// TIA Portal V15 export
// export: Created 2018-05-29T12:25:38.1552518Z, ExportSetting WithDefaults, DisplayName Totally Integrated Automation Portal, DisplayVersion V15, DisplayName STEP 7 Professional, DisplayVersion V15, DisplayName WinCC Professional, DisplayVersion V15, DisplayName TIA Portal Openness, DisplayVersion V15
FUNCTION "LIC006_fc" : Void   // FC1, STL
TITLE = LIC006_fc
{ S7_Optimized_Access := 'TRUE' }
VERSION : 0.1
// test
// stored: AutoNumber true, UDAEnableTagReadback false
BEGIN

NETWORK
TITLE = Change PID Setpoints
// The phase FBs write on the operator setpoints of the PID-controller
// To avoid that the setpoints are always overwritten (and blocking operator control)
// we use pulses generated by the phase to set the setpoints only at specific moments
// i_fOCmdSP (setpoint)
// i_fOCmdMANOP (output)
      CALL  "BST_PIDAIN_400", "DB";


//Write the Operator_Setpoint
      A     "LIC006_sp".Set_SP;
      JCN   J001;

      L     "LIC006_sp".Operator_Setpoint;
      T     "LIC006".i_fOCmdSP;

J001: NOP   0;


//Write the Output_Value
      A     "LIC006_sp".Set_Output;
      JCN   J002;

      L     "LIC006_sp".Output_Value;
      T     "LIC006".i_fOCmdMANOP;

J002: NOP   0;



NETWORK
TITLE = Main
// comment: PLC1


//Call the CM FB with the corresponding DB instance
END_FUNCTION
